# EPICS substitutions: viocs/ts_ps/ts_psApp/Db/bend.substitutions
file "db/individual.db" {
    pattern { family, pos }
        { "BEND", "01" }
        { "BEND", "02" }
        { "BEND", "03" }
}
